FUNCTION_BLOCK ABSTRACT FB_BaseSensor IMPLEMENTS I_SafetySensor
VAR
    _rValue         : REAL ;
    _eStatus        : E_SensorStatus := E_SensorStatus.SENSOR_OK;
    _bAlarm         : BOOL := FALSE;
    _bFault         : BOOL := FALSE;
    _sLocation      : STRING := '';
END_VAR
VAR_INPUT
    rRawValue       : REAL := 0.0;      // simulated input — HMI slider
    bSimFault       : BOOL := FALSE;    // simulate sensor fault
END_VAR

{warning 'add method implementation '}
METHOD GetReading : REAL
GetReading := _rValue;
END_METHOD

{warning 'add method implementation '}
METHOD GetStatus : E_SensorStatus
GetStatus := _eStatus;
END_METHOD

{warning 'add method implementation '}
METHOD IsAlarm : BOOL
IsAlarm := _bAlarm;
END_METHOD

{warning 'add method implementation '}
METHOD IsFault : BOOL
IsFault := _bFault;
END_METHOD

{warning 'add method implementation '}
METHOD Reset
_bAlarm  := FALSE;
_bFault  := FALSE;
_eStatus := E_SensorStatus.SENSOR_OK;
END_METHOD

METHOD ABSTRACT Validate 
VAR_INPUT
END_VAR
END_METHOD

END_FUNCTION_BLOCK

(* stored: Version 1.1.0.1, ProductVersion 3.1.4024.16
   POU FB_BaseSensor: Id {f8879f13-8d0d-4f5e-a5fc-a23b3f6e36a1}, SpecialFunc None
   Method GetReading: Id {d37d12cd-1892-449a-b1d0-fe9e0adc7e0a}
   Method GetStatus: Id {93044ec1-55c7-427a-9ef9-35d8e1c24c73}
   Method IsAlarm: Id {14b8bc43-12b3-458a-a170-2ed52d722756}
   Method IsFault: Id {26f1683c-35e7-4d7b-97c1-b465cd0e12ac}
   Method Reset: Id {596d7f60-2e43-4ed1-90b2-f66e781faa68}
   Method Validate: Id {3ecf1198-f7af-498b-95ca-a847b9bfd83c} *)
